Universal Robots PolyScope program: rs3_task_peter.urp

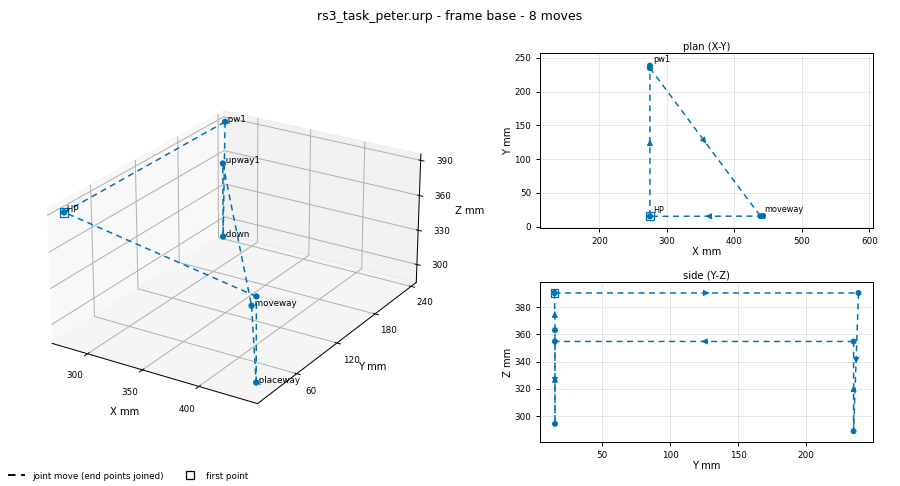
[picture p0: tool path of rs3_task_peter.urp in frame base, 8 of 8 moves have a stored position in this frame; points joined in program order, loops and branches not executed]
Program rs3_task_peter (installation=default directory=/programs/palletizing createdIn=5.11.9.1010452 lastSavedIn=5.11.9.1010452 robotSerialNumber=20225200364)
Calibrated DH parameters: a=[0.00002, -0.569483, -0.54992, -0.00001, -0.000036, 0]; d=[0.180894, -146.691669, 192.918669, -46.053088, 0.119778, 0.115602]; alpha=[1.571425, -0.001534, 0.003359, 1.568739, -1.571477, 0]; deltaTheta=[0, 0.376258, -0.101074, -0.275185, -0.000002, 0]
Robot Program (runOnlyOnce=false)
  MoveJ speed 60 deg/s, acceleration 80 deg/s^2 (useActiveTCP=true) feature=Base
    Waypoint HP: TCP in base x=274.852 y=15.069 z=390.532 mm, rx=2.2312 ry=-2.2053 rz=0.0033 rad; joints [42.51, -73.428, -133.962, -242.896, -90.073, -137.934] deg
    Waypoint pw1: TCP in base x=274.853 y=238.502 z=390.527 mm, rx=2.2314 ry=-2.2053 rz=0.0033 rad; joints [69.565, -84.808, -125.205, -240.303, -90.181, -110.867] deg
    Waypoint down: TCP in base x=274.869 y=234.901 z=288.915 mm, rx=2.2312 ry=-2.2054 rz=0.0033 rad; joints [69.354, -91.732, -131.251, -227.334, -90.157, -111.026] deg
    URCap RG Grip (OnRobot, OnRobot A/S) dataModel(rg-target-force=40.0, rg-target-width=0.08, Variable(key=on_return, variable(name=on_return)))
    Waypoint upway1: TCP in base x=274.869 y=234.899 z=354.873 mm, rx=2.2312 ry=-2.2053 rz=0.0034 rad; joints [69.342, -86.75, -127.669, -235.902, -90.175, -111.068] deg
    Waypoint moveway: TCP in base x=438.4 y=15.391 z=354.877 mm, rx=2.2312 ry=-2.2053 rz=0.0033 rad; joints [25.468, -94.674, -119.592, -235.972, -89.972, -154.938] deg
    Waypoint placeway: TCP in base x=442.45 y=15.425 z=294.322 mm, rx=2.2312 ry=-2.2054 rz=0.0034 rad; joints [25.233, -99.083, -122.143, -229.006, -89.956, -155.148] deg
    URCap RG Grip (OnRobot, OnRobot A/S) dataModel(rg-target-force=40.0, rg-target-width=0.1)
    Waypoint upway2: TCP in base x=442.427 y=15.423 z=363.179 mm, rx=2.2312 ry=-2.2053 rz=0.0033 rad; joints [25.227, -94.571, -118.704, -236.962, -89.972, -155.184] deg
    Waypoint HP: TCP in base x=274.852 y=15.069 z=390.532 mm, rx=2.2312 ry=-2.2053 rz=0.0033 rad; joints [42.51, -73.428, -133.962, -242.896, -90.073, -137.934] deg
    Halt
